% RSLogix 500 project P7_ASHLEY_J.RSS, saved by version 8.30.00.16 %
PROJECT "UNTITLED"    % processor: Bul.1763 MicroLogix 1100 Series B %

PROGRAM FILES
  LAD 2 "MAIN"  4 rungs
  LAD 3 "IO"  4 rungs
  LAD 4 "CALIBRATE"  10 rungs
  LAD 5 "CONTROLS"  11 rungs

DATA FILES
  O0 OUTPUT  4 elements
  I1 INPUT  6 elements
  S2 STATUS  66 elements
  B3 BINARY  10 elements
  T4 TIMER  4 elements
  C5 COUNTER  2 elements
  R6 CONTROL  1 elements
  N7 INTEGER  1 elements
  F8 FLOAT  16 elements

LADDER 2 "MAIN"
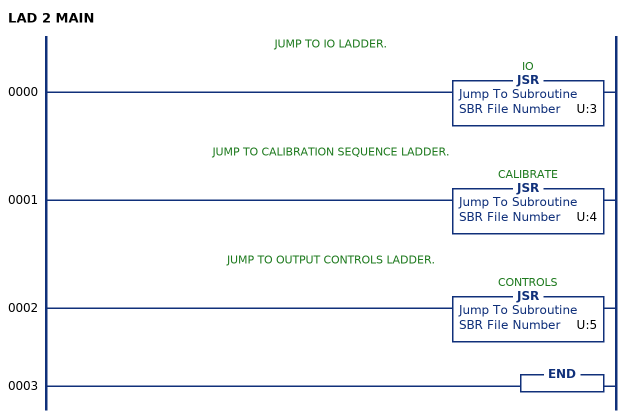
% Rung: 0 %
% JUMP TO IO LADDER. %
SOR JSR U:3 EOR
%   U:3  "IO" %
% Rung: 1 %
% JUMP TO CALIBRATION SEQUENCE LADDER. %
SOR JSR U:4 EOR
%   U:4  "CALIBRATE" %
% Rung: 2 %
% JUMP TO OUTPUT CONTROLS LADDER. %
SOR JSR U:5 EOR
%   U:5  "CONTROLS" %
% Rung: 3 %
SOR END EOR

LADDER 3 "IO"
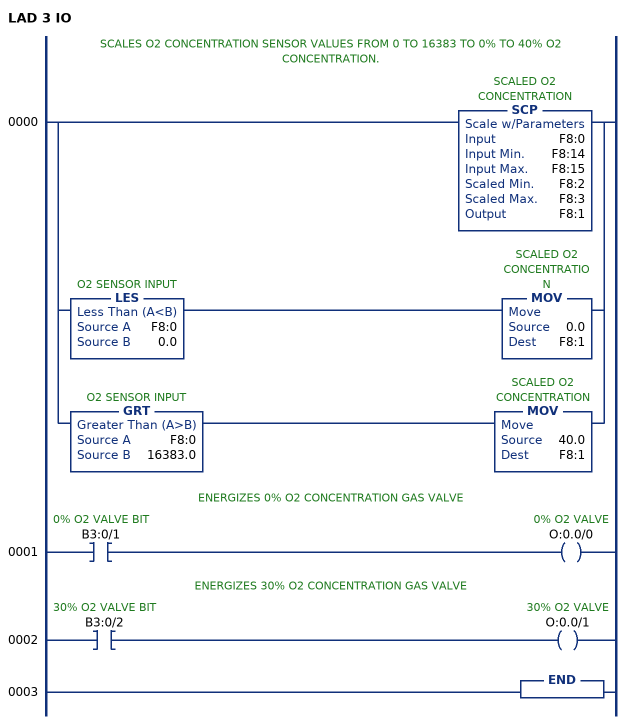
% Rung: 0 %
% SCALES O2 CONCENTRATION SENSOR VALUES FROM 0 TO 16383 TO 0% TO 40% O2 CONCENTRATION. %
SOR BST SCP F8:0 F8:14 F8:15 F8:2 F8:3 F8:1 NXB LES F8:0 0.0 MOV 0.0 F8:1 NXB GRT F8:0 16383.0 MOV 40.0 F8:1 BND EOR
%   F8:0  "O2 SENSOR INPUT" %
%   F8:14  "INPUT MIN" %
%   F8:15  "INPUT MAX" %
%   F8:2  "O2 SENSOR SCALED INPUT MIN" %
%   F8:3  "O2 SENSOR SCALED INPUT MAX" %
%   F8:1  "SCALED O2 CONCENTRATION" %
% Rung: 1 %
% ENERGIZES 0% O2 CONCENTRATION GAS VALVE %
SOR XIC B3:0/1 OTE O:0.0/0 EOR
%   B3:0/1  "0% O2 VALVE BIT" %
%   O:0.0/0  "0% O2 VALVE" %
% Rung: 2 %
% ENERGIZES 30% O2 CONCENTRATION GAS VALVE %
SOR XIC B3:0/2 OTE O:0.0/1 EOR
%   B3:0/2  "30% O2 VALVE BIT" %
%   O:0.0/1  "30% O2 VALVE" %
% Rung: 3 %
SOR END EOR

LADDER 4 "CALIBRATE"
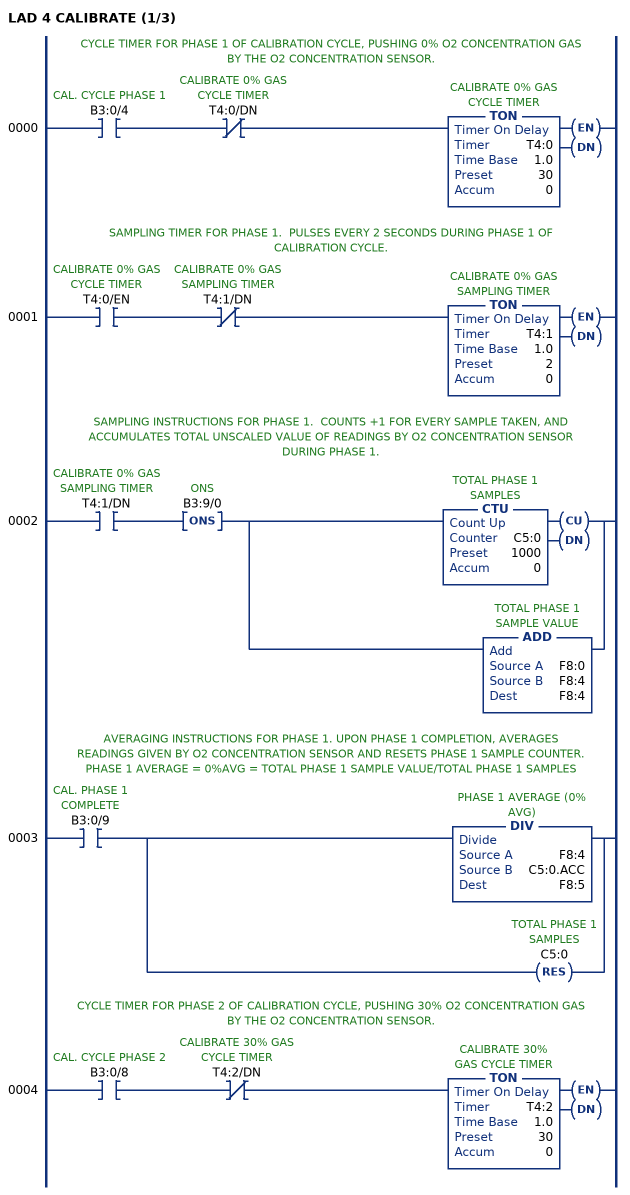
% Rung: 0 %
% CYCLE TIMER FOR PHASE 1 OF CALIBRATION CYCLE, PUSHING 0% O2 CONCENTRATION GAS BY THE O2 CONCENTRATION SENSOR. %
SOR XIC B3:0/4 XIO T4:0/DN TON T4:0 1.0 30 0 EOR
%   B3:0/4  "CAL. CYCLE PHASE 1" %
%   T4:0  "CALIBRATE 0% GAS CYCLE TIMER" %
% Rung: 1 %
% SAMPLING TIMER FOR PHASE 1.  PULSES EVERY 2 SECONDS DURING PHASE 1 OF CALIBRATION CYCLE. %
SOR XIC T4:0/EN XIO T4:1/DN TON T4:1 1.0 2 0 EOR
%   T4:0  "CALIBRATE 0% GAS CYCLE TIMER" %
%   T4:1  "CALIBRATE 0% GAS SAMPLING TIMER" %
% Rung: 2 %
% SAMPLING INSTRUCTIONS FOR PHASE 1.  COUNTS +1 FOR EVERY SAMPLE TAKEN, AND ACCUMULATES TOTAL UNSCALED VALUE OF READINGS BY O2 CONCENTRATION SENSOR DURING PHASE 1. %
SOR XIC T4:1/DN ONS B3:9/0 BST CTU C5:0 1000 0 NXB ADD F8:0 F8:4 F8:4 BND EOR
%   T4:1  "CALIBRATE 0% GAS SAMPLING TIMER" %
%   B3:9/0  "ONS" %
%   C5:0  "TOTAL PHASE 1 SAMPLES" %
%   F8:0  "O2 SENSOR INPUT" %
%   F8:4  "TOTAL PHASE 1 SAMPLE VALUE" %
% Rung: 3 %
% AVERAGING INSTRUCTIONS FOR PHASE 1. UPON PHASE 1 COMPLETION, AVERAGES READINGS GIVEN BY O2 CONCENTRATION SENSOR AND RESETS PHASE 1 SAMPLE COUNTER. PHASE 1 AVERAGE = 0%AVG = TOTAL PHASE 1 SAMPLE VALUE/TOTAL PHASE 1 SAMPLES %
SOR XIC B3:0/9 BST DIV F8:4 C5:0.ACC F8:5 NXB RES C5:0 BND EOR
%   B3:0/9  "CAL. PHASE 1 COMPLETE" %
%   F8:4  "TOTAL PHASE 1 SAMPLE VALUE" %
%   C5:0  "TOTAL PHASE 1 SAMPLES" %
%   F8:5  "PHASE 1 AVERAGE (0% AVG)" %
% Rung: 4 %
% CYCLE TIMER FOR PHASE 2 OF CALIBRATION CYCLE, PUSHING 30% O2 CONCENTRATION GAS BY THE O2 CONCENTRATION SENSOR. %
SOR XIC B3:0/8 XIO T4:2/DN TON T4:2 1.0 30 0 EOR
%   B3:0/8  "CAL. CYCLE PHASE 2" %
%   T4:2  "CALIBRATE 30% GAS CYCLE TIMER" %

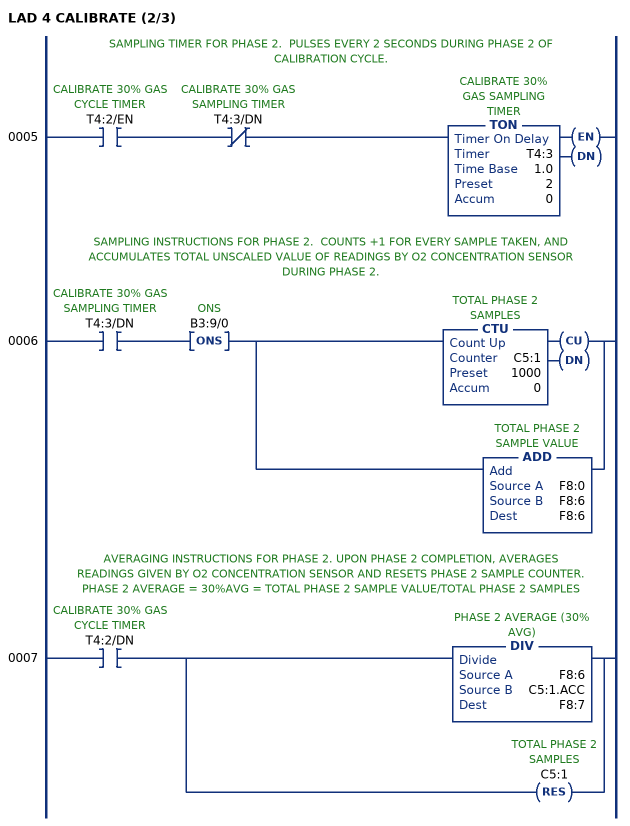
% Rung: 5 %
% SAMPLING TIMER FOR PHASE 2.  PULSES EVERY 2 SECONDS DURING PHASE 2 OF CALIBRATION CYCLE. %
SOR XIC T4:2/EN XIO T4:3/DN TON T4:3 1.0 2 0 EOR
%   T4:2  "CALIBRATE 30% GAS CYCLE TIMER" %
%   T4:3  "CALIBRATE 30% GAS SAMPLING TIMER" %
% Rung: 6 %
% SAMPLING INSTRUCTIONS FOR PHASE 2.  COUNTS +1 FOR EVERY SAMPLE TAKEN, AND ACCUMULATES TOTAL UNSCALED VALUE OF READINGS BY O2 CONCENTRATION SENSOR DURING PHASE 2. %
SOR XIC T4:3/DN ONS B3:9/0 BST CTU C5:1 1000 0 NXB ADD F8:0 F8:6 F8:6 BND EOR
%   T4:3  "CALIBRATE 30% GAS SAMPLING TIMER" %
%   B3:9/0  "ONS" %
%   C5:1  "TOTAL PHASE 2 SAMPLES" %
%   F8:0  "O2 SENSOR INPUT" %
%   F8:6  "TOTAL PHASE 2 SAMPLE VALUE" %
% Rung: 7 %
% AVERAGING INSTRUCTIONS FOR PHASE 2. UPON PHASE 2 COMPLETION, AVERAGES READINGS GIVEN BY O2 CONCENTRATION SENSOR AND RESETS PHASE 2 SAMPLE COUNTER. PHASE 2 AVERAGE = 30%AVG = TOTAL PHASE 2 SAMPLE VALUE/TOTAL PHASE 2 SAMPLES %
SOR XIC T4:2/DN BST DIV F8:6 C5:1.ACC F8:7 NXB RES C5:1 BND EOR
%   T4:2  "CALIBRATE 30% GAS CYCLE TIMER" %
%   F8:6  "TOTAL PHASE 2 SAMPLE VALUE" %
%   C5:1  "TOTAL PHASE 2 SAMPLES" %
%   F8:7  "PHASE 2 AVERAGE (30% AVG)" %

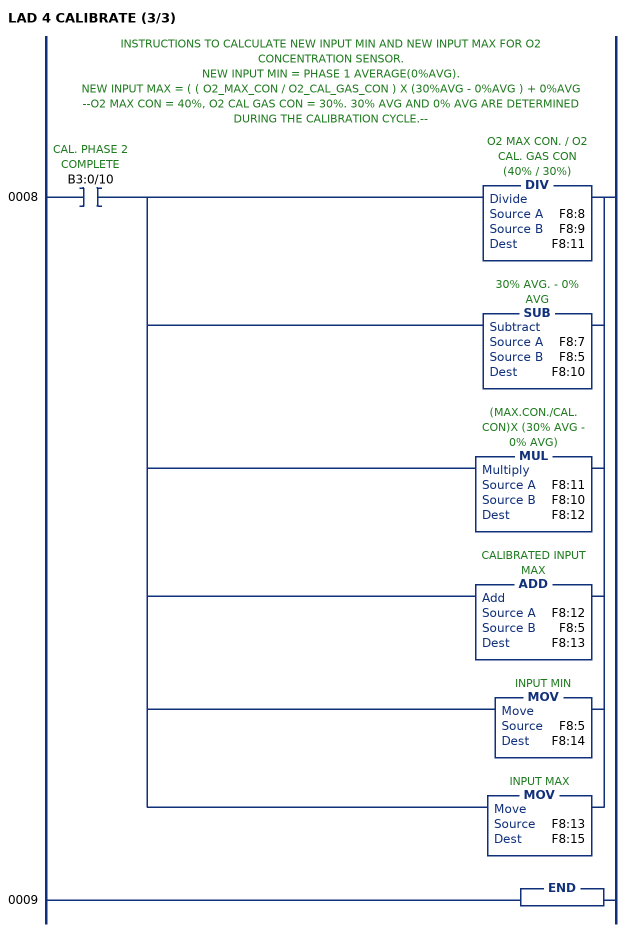
% Rung: 8 %
% INSTRUCTIONS TO CALCULATE NEW INPUT MIN AND NEW INPUT MAX FOR O2 CONCENTRATION SENSOR.
% NEW INPUT MIN = PHASE 1 AVERAGE(0%AVG).
% NEW INPUT MAX = ( ( O2_MAX_CON / O2_CAL_GAS_CON ) X (30%AVG - 0%AVG ) + 0%AVG
% --O2 MAX CON = 40%, O2 CAL GAS CON = 30%. 30% AVG AND 0% AVG ARE DETERMINED DURING THE CALIBRATION CYCLE.-- %
SOR XIC B3:0/10 BST DIV F8:8 F8:9 F8:11 NXB SUB F8:7 F8:5 F8:10 NXB MUL F8:11 F8:10 F8:12 NXB ADD F8:12 F8:5 F8:13 NXB MOV F8:5 F8:14 NXB MOV F8:13 F8:15 BND EOR
%   B3:0/10  "CAL. PHASE 2 COMPLETE" %
%   F8:8  "O2 MAX CON." %
%   F8:9  "CAL. GAS CON" %
%   F8:11  "O2 MAX CON. / O2 CAL. GAS CON (40% / 30%)" %
%   F8:7  "PHASE 2 AVERAGE (30% AVG)" %
%   F8:5  "PHASE 1 AVERAGE (0% AVG)" %
%   F8:10  "30% AVG. - 0% AVG" %
%   F8:12  "(MAX.CON./CAL.CON)X (30% AVG - 0% AVG)" %
%   F8:13  "CALIBRATED INPUT MAX" %
%   F8:14  "INPUT MIN" %
%   F8:15  "INPUT MAX" %
% Rung: 9 %
SOR END EOR

LADDER 5 "CONTROLS"
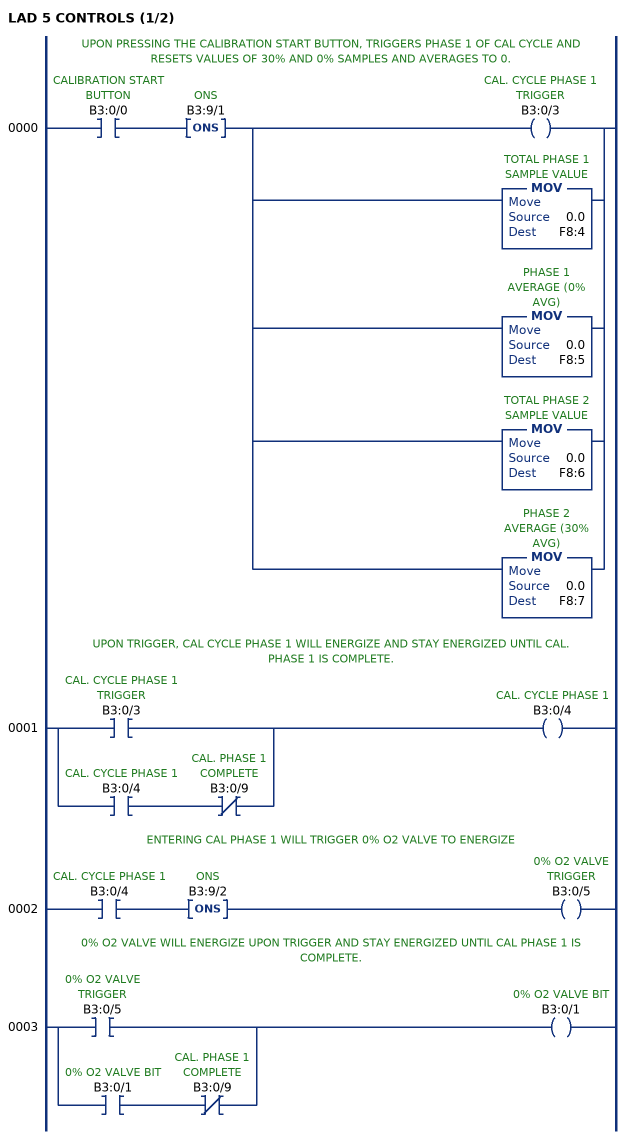
% Rung: 0 %
% UPON PRESSING THE CALIBRATION START BUTTON, TRIGGERS PHASE 1 OF CAL CYCLE AND RESETS VALUES OF 30% AND 0% SAMPLES AND AVERAGES TO 0. %
SOR XIC B3:0/0 ONS B3:9/1 BST OTE B3:0/3 NXB MOV 0.0 F8:4 NXB MOV 0.0 F8:5 NXB MOV 0.0 F8:6 NXB MOV 0.0 F8:7 BND EOR
%   B3:0/0  "CALIBRATION START BUTTON" %
%   B3:9/1  "ONS" %
%   B3:0/3  "CAL. CYCLE PHASE 1 TRIGGER" %
%   F8:4  "TOTAL PHASE 1 SAMPLE VALUE" %
%   F8:5  "PHASE 1 AVERAGE (0% AVG)" %
%   F8:6  "TOTAL PHASE 2 SAMPLE VALUE" %
%   F8:7  "PHASE 2 AVERAGE (30% AVG)" %
% Rung: 1 %
% UPON TRIGGER, CAL CYCLE PHASE 1 WILL ENERGIZE AND STAY ENERGIZED UNTIL CAL. PHASE 1 IS COMPLETE. %
SOR BST XIC B3:0/3 NXB XIC B3:0/4 XIO B3:0/9 BND OTE B3:0/4 EOR
%   B3:0/3  "CAL. CYCLE PHASE 1 TRIGGER" %
%   B3:0/4  "CAL. CYCLE PHASE 1" %
%   B3:0/9  "CAL. PHASE 1 COMPLETE" %
% Rung: 2 %
% ENTERING CAL PHASE 1 WILL TRIGGER 0% O2 VALVE TO ENERGIZE %
SOR XIC B3:0/4 ONS B3:9/2 OTE B3:0/5 EOR
%   B3:0/4  "CAL. CYCLE PHASE 1" %
%   B3:9/2  "ONS" %
%   B3:0/5  "0% O2 VALVE TRIGGER" %
% Rung: 3 %
% 0% O2 VALVE WILL ENERGIZE UPON TRIGGER AND STAY ENERGIZED UNTIL CAL PHASE 1 IS COMPLETE. %
SOR BST XIC B3:0/5 NXB XIC B3:0/1 XIO B3:0/9 BND OTE B3:0/1 EOR
%   B3:0/5  "0% O2 VALVE TRIGGER" %
%   B3:0/1  "0% O2 VALVE BIT" %
%   B3:0/9  "CAL. PHASE 1 COMPLETE" %

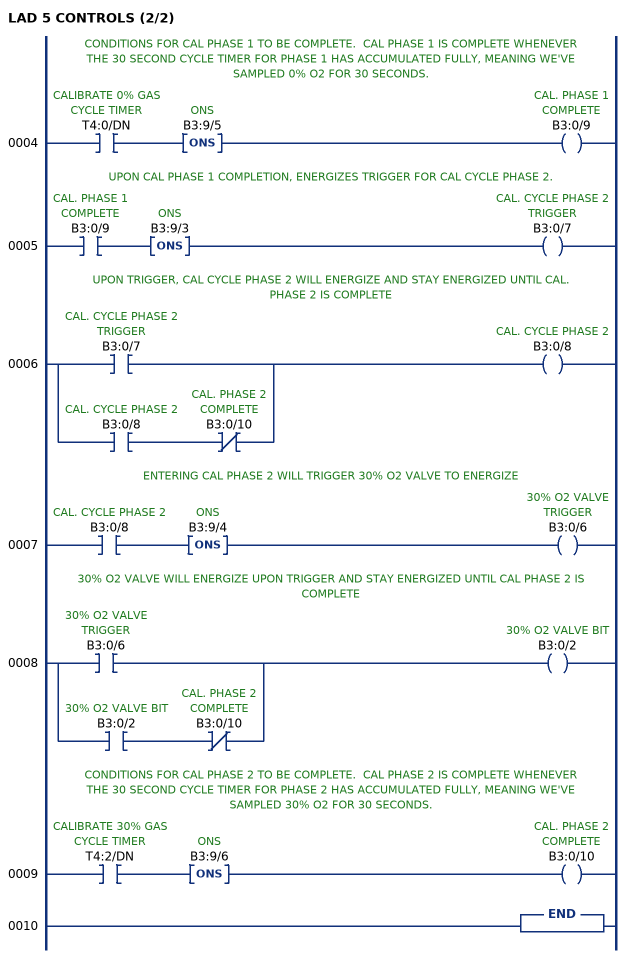
% Rung: 4 %
% CONDITIONS FOR CAL PHASE 1 TO BE COMPLETE.  CAL PHASE 1 IS COMPLETE WHENEVER THE 30 SECOND CYCLE TIMER FOR PHASE 1 HAS ACCUMULATED FULLY, MEANING WE'VE SAMPLED 0% O2 FOR 30 SECONDS. %
SOR XIC T4:0/DN ONS B3:9/5 OTE B3:0/9 EOR
%   T4:0  "CALIBRATE 0% GAS CYCLE TIMER" %
%   B3:9/5  "ONS" %
%   B3:0/9  "CAL. PHASE 1 COMPLETE" %
% Rung: 5 %
% UPON CAL PHASE 1 COMPLETION, ENERGIZES TRIGGER FOR CAL CYCLE PHASE 2. %
SOR XIC B3:0/9 ONS B3:9/3 OTE B3:0/7 EOR
%   B3:0/9  "CAL. PHASE 1 COMPLETE" %
%   B3:9/3  "ONS" %
%   B3:0/7  "CAL. CYCLE PHASE 2 TRIGGER" %
% Rung: 6 %
% UPON TRIGGER, CAL CYCLE PHASE 2 WILL ENERGIZE AND STAY ENERGIZED UNTIL CAL. PHASE 2 IS COMPLETE %
SOR BST XIC B3:0/7 NXB XIC B3:0/8 XIO B3:0/10 BND OTE B3:0/8 EOR
%   B3:0/7  "CAL. CYCLE PHASE 2 TRIGGER" %
%   B3:0/8  "CAL. CYCLE PHASE 2" %
%   B3:0/10  "CAL. PHASE 2 COMPLETE" %
% Rung: 7 %
% ENTERING CAL PHASE 2 WILL TRIGGER 30% O2 VALVE TO ENERGIZE %
SOR XIC B3:0/8 ONS B3:9/4 OTE B3:0/6 EOR
%   B3:0/8  "CAL. CYCLE PHASE 2" %
%   B3:9/4  "ONS" %
%   B3:0/6  "30% O2 VALVE TRIGGER" %
% Rung: 8 %
% 30% O2 VALVE WILL ENERGIZE UPON TRIGGER AND STAY ENERGIZED UNTIL CAL PHASE 2 IS COMPLETE %
SOR BST XIC B3:0/6 NXB XIC B3:0/2 XIO B3:0/10 BND OTE B3:0/2 EOR
%   B3:0/6  "30% O2 VALVE TRIGGER" %
%   B3:0/2  "30% O2 VALVE BIT" %
%   B3:0/10  "CAL. PHASE 2 COMPLETE" %
% Rung: 9 %
% CONDITIONS FOR CAL PHASE 2 TO BE COMPLETE.  CAL PHASE 2 IS COMPLETE WHENEVER THE 30 SECOND CYCLE TIMER FOR PHASE 2 HAS ACCUMULATED FULLY, MEANING WE'VE SAMPLED 30% O2 FOR 30 SECONDS. %
SOR XIC T4:2/DN ONS B3:9/6 OTE B3:0/10 EOR
%   T4:2  "CALIBRATE 30% GAS CYCLE TIMER" %
%   B3:9/6  "ONS" %
%   B3:0/10  "CAL. PHASE 2 COMPLETE" %
% Rung: 10 %
SOR END EOR

OTHER DOCUMENTED ADDRESSES
  B3:8/0  "TESTING INTERLOCK"

DATA TABLE (non-zero values as saved)
DATA T4
% .PRE .ACC %
% T4:0 % 30 0
% T4:1 % 2 0
% T4:2 % 30 0
% T4:3 % 2 0
DATA C5
% .PRE .ACC %
% C5:0 % 1000 0
% C5:1 % 1000 0
DATA F8
% F8:0 % 0 0 0 40 0
% F8:5 % 0 0 0 40 30
% F8:15 % 16383
